Staubli VAL3: writeIntValue.pgx

public program writeIntValue(num x_nCamID (dimensions=1), string x_sCellNumber (dimensions=1), num x_nValue (dimensions=1), bool& x_bError[] (dimensions=1))
  local string l_sCell
  local bool l_bIsOk
begin
  //-----------------------------------------------------------------------
  //Header begin
  //Description of program
  //  Sets the control contained in a cell (x_sCellNumber) to the specified
  //  integer value (x_nValue).
  //  The target cell of the writing operation in the Cognex spreadsheet must
  //  be of the EditInt type.
  //
  //Input parameters
  //  num x_nCamID :
  //    role : camera's ID
  //  string x_sCellNumber :
  //    role : The column letter and the row number of the cell value to get.
  //    possible values : - column letter : (A to Z)
  //                      - row number : (000 to 399)
  //  num x_nValue :
  //    role : value to writing in the cell
  //
  //Output parameters
  //  bool x_bError :
  //    role : returns true if an error occurred and false otherwise
  //
  //Examples
  //  call writeIntValue(nCamID,"C6",8,l_bError)
  //
  //History
  //  Creation : 19-05-08 - f.Rob
  //Header end
  //-----------------------------------------------------------------------

  x_bError=true
  call checkCellFormat(x_nCamID,x_sCellNumber,l_bIsOk)
  if l_bIsOk
    nProgram[x_nCamID]=10
    call sendCommand(x_nCamID,"SI"+x_sCellNumber+toString("0.0",roundDown(x_nValue)),x_bError)
  endIf
end
